TEXTLIST TextList_Recipe
  1 = '1'
  2 = '2'
  3 = '3'
  4 = '4'
  5 = '5'
  6 = '6'
   = ''
END_TEXTLIST

(* stored: Version 1.1.0.1, ProductVersion 3.1.4024.12
   TextList TextList_Recipe: Id {8be698d1-ead9-44a9-89f7-79818a36ae55} *)
